FUNCTION_BLOCK FB_Impulse
VAR_INPUT
	bInputs			:	ARRAY[0..nSize] OF BOOL;	//Input Schalter oder Taster
	bInputSecLoop	:	BOOL := FALSE;				//Input für Security Loop
	bR_Trig			:	BOOL := TRUE;				//Steigende Flanke? Wenn FALSE = Fallend
	tHigh			:	TIME;						//Zeit (ms) für High
	tDelay			:	TIME := T#0MS;				//Verzögerungszeit (ms) zwischen den Impulsen									
END_VAR
VAR_OUTPUT
	bOut			:	BOOL;
END_VAR
VAR_IN_OUT
	bInputHA		:	BOOL;
END_VAR
VAR CONSTANT
	nSize 			:	UINT := 5; 					//Maximale Anzahl Eingänge
END_VAR
VAR
	fbRtrig			:	ARRAY[0..nSize] OF R_TRIG;
	fbFtrig			:	ARRAY[0..nSize] OF F_TRIG;
	
	fbRtrigInit		:	R_TRIG;
	
	Idx				:	UINT;
	bTrigger		:	BOOL;
	
	tpPulse			:	TP;
	tofDelay		:	TOF;
	
END_VAR
VAR_TEMP

END_VAR



//--------------------------------------Notfall Toggle
fbRtrigInit(CLK:= bInputSecLoop, Q=> );
tpPulse(IN := bOut, PT := tHigh);
tofDelay(IN := bOut, PT := tHigh);

IF bInputSecLoop THEN
		
	IF fbRtrigInit.Q THEN
		bOut	:= TRUE;
	END_IF
	
	IF NOT tpPulse.Q THEN
		bOut := FALSE;
	END_IF
	
	IF NOT tofDelay.Q THEN
		bOut := TRUE;
	END_IF	
	
ELSE //----------------------------------Normaler Impuls
	bTrigger 	:= FALSE;

	//Init alle Flankentrigger und Frage diese ab
	FOR Idx := 0 TO nSize DO
	
		IF bR_Trig THEN
		
			fbRtrig[Idx](CLK:= bInputs[Idx], Q=> );
			bTrigger := bTrigger OR fbRtrig[Idx].Q;
	
		ELSE
	
			fbFtrig[Idx](CLK:= bInputs[Idx], Q=> );
			bTrigger := bTrigger OR fbFtrig[Idx].Q;
	
		END_IF
	
	END_FOR
	
	bTrigger := bTrigger OR bInputHA;
	
	IF NOT tofDelay.Q THEN
		tpPulse(IN := bTrigger, PT := tHigh);
	END_IF

	IF tpPulse.Q THEN
		bOut 		:= TRUE;
		bInputHA 	:= TRUE;
	ELSE
		bOut 		:= FALSE;
		bInputHA	:= FALSE;
		tofDelay(IN := bOut, PT := tDelay);
	END_IF
	
END_IF

END_FUNCTION_BLOCK

(* stored: Version 1.1.0.1, ProductVersion 3.1.4024.4
   POU FB_Impulse: Id {16b34e2a-1064-4431-9540-1d9a54fc44a9}, SpecialFunc None *)
